// TwinCAT 3 PLC project Library
// Title: MTP
// Company: Zerlauth
// Author: Peter Zerlauth
// ProjectVersion: 0.0.0.0
// Description: Module Type Package MTP
// ProgramVersion: 3.1.4024.0
// libraries:
//   Tc2_Standard, * (Beckhoff Automation GmbH)
//   Tc2_System, * (Beckhoff Automation GmbH)
//   Tc2_Utilities, * (Beckhoff Automation GmbH)
// project tree:
//   Component/Event/ E_Event.TcDUT, FB_Event.TcPOU, I_Event.TcIO, ST_Event.TcDUT
//   Component/ E_Request.TcDUT, E_State.TcDUT, FB_Component.TcPOU, I_Component.TcIO, ST_Component.TcDUT (not stored)
//   Component/Info/ FB_Info.TcPOU, I_Info.TcIO (not stored)
//   Component/Observer/ FB_Observer.TcPOU, I_Observer.TcIO
//   List/ FB_ListComponent.TcPOU, FB_ListObject.TcPOU, FB_ListString.TcPOU, I_ListComponent.TcIO, I_ListObject.TcIO, I_ListString.TcIO (not stored)
//   Logger/ FB_ListLogger.TcPOU, I_Logger.TcIO
//   Object/ I_Object.TcIO
//   Sequence/ FB_Sequence.TcPOU (not stored), I_Sequence.TcIO (not stored)
// (motion and I/O tree: see PLC project example)
// real-time tasks:
//   TASK plcTask1: cycle T#1000ms, priority 20, ADS port 350

// ---- Component/Event/E_Event.TcDUT
{attribute 'qualified_only'}
{attribute 'strict'}
TYPE E_Event :
(
	Verbose			:= 0,
	Debug			:= 1,
	Information		:= 2,
	Warning			:= 3,
	Error			:= 4
);
END_TYPE

// ---- Component/Event/ST_Event.TcDUT
TYPE ST_Event :
STRUCT
	Timestamp:   	ULINT;
	ID:				UDINT;
	Message:		STRING(255);
	Arguments:		STRING(255);
END_STRUCT
END_TYPE

// ---- Component/E_Request.TcDUT
{attribute 'qualified_only'}
{attribute 'strict'}
TYPE E_Request :
(
    Undefined   := 0,
	Reset       := 1,
    Start       := 2,
    Pause       := 4,	
    Hold      	:= 8,
	Complete	:= 16,	
    Stop        := 32,
	Abort       := 64
);
END_TYPE

// ---- Component/E_State.TcDUT
{attribute 'qualified_only'}
{attribute 'strict'}
TYPE E_State :
(
	Undefined		:= 0,
	Clearing		:= 1,
	Stopped			:= 2,
	Starting		:= 3,
	Idle			:= 4,
	Suspend			:= 5,
	Execute			:= 6,
	Stopping		:= 7,
	Aborting		:= 8,
	Aborted			:= 9,
	Holding			:= 10,
	Held			:= 11,
	Unholding		:= 12,
	Suspending		:= 13,
	Unsuspending	:= 14,
	Resetting		:= 15,
	Completing		:= 16,
	Complete		:= 17
);
END_TYPE

// ---- Component/Event/I_Event.TcIO
INTERFACE I_Event EXTENDS I_Object

METHOD PUBLIC M_Abort : BOOL
VAR_INPUT
	Message:				STRING(255);
	ID:						UDINT;
END_VAR
END_METHOD

METHOD PUBLIC M_Debug : BOOL
VAR_INPUT
	Message:				STRING(255);
END_VAR
END_METHOD

METHOD PUBLIC M_Information : BOOL
VAR_INPUT
	Message:				STRING(255);
	ID:						UDINT;
END_VAR
END_METHOD

METHOD PUBLIC M_Stop : BOOL
VAR_INPUT
	Message:				STRING(255);
	ID:						UDINT;
END_VAR
END_METHOD

METHOD PUBLIC M_Warning : BOOL
VAR_INPUT
	Message:				STRING(255);
	ID:						UDINT;
END_VAR
END_METHOD

PROPERTY PUBLIC P_Logger : I_Logger
GET
END_GET
SET
END_SET
END_PROPERTY

END_INTERFACE

// ---- Component/I_Component.TcIO
INTERFACE I_Component EXTENDS I_Object

METHOD PUBLIC M_Request : BOOL
VAR_INPUT
	eRequest:	E_Request;
END_VAR
END_METHOD

PROPERTY PUBLIC P_Event : I_Event
GET
END_GET
END_PROPERTY

PROPERTY PUBLIC P_Info : I_Info
GET
END_GET
END_PROPERTY

PROPERTY PUBLIC P_Observer : I_Observer
GET
END_GET
END_PROPERTY

END_INTERFACE

// ---- Component/Observer/I_Observer.TcIO
INTERFACE I_Observer

METHOD M_Attach : BOOL
VAR_INPUT
	Object: 	I_Component;
END_VAR
END_METHOD

METHOD M_Detach : BOOL
VAR_INPUT
	Object: 	I_Component;
END_VAR
END_METHOD

METHOD M_Notify : BOOL
VAR_INPUT
	eRequest:		E_Request;
END_VAR
END_METHOD

END_INTERFACE

// ---- List/I_ListComponent.TcIO
INTERFACE I_ListComponent

METHOD M_Add : BOOL
VAR_INPUT
	Object: 	I_Component;
END_VAR
END_METHOD

METHOD M_Clear : BOOL
END_METHOD

METHOD M_Find : DINT
VAR_INPUT
	Object: 	I_Component;
END_VAR
END_METHOD

METHOD M_Index : I_Component
VAR_INPUT
	Index: 	DINT;
END_VAR
END_METHOD

METHOD M_Remove : BOOL
VAR_INPUT
	Object: 	I_Component;
END_VAR
END_METHOD

METHOD PUBLIC M_Request : BOOL
VAR_INPUT
	eRequest:		E_Request;
END_VAR
END_METHOD

PROPERTY P_Length : DINT
GET
END_GET
END_PROPERTY

END_INTERFACE

// ---- List/I_ListObject.TcIO
INTERFACE I_ListObject

METHOD M_Add : BOOL
VAR_INPUT
	Object: 	I_Object;
END_VAR
END_METHOD

METHOD M_Clear : BOOL
END_METHOD

METHOD M_Find : DINT
VAR_INPUT
	Object: 	I_Object;
END_VAR
END_METHOD

METHOD M_Index : I_Object
VAR_INPUT
	Index: 	DINT;
END_VAR
END_METHOD

METHOD M_Remove : BOOL
VAR_INPUT
	Object: 	I_Object;
END_VAR
END_METHOD

PROPERTY P_Length : DINT
GET
END_GET
END_PROPERTY

END_INTERFACE

// ---- Logger/I_Logger.TcIO
INTERFACE I_Logger EXTENDS I_Object

METHOD PUBLIC M_Log
VAR_INPUT
	stEvent:		ST_Event;
END_VAR
END_METHOD

END_INTERFACE

// ---- Object/I_Object.TcIO
INTERFACE I_Object EXTENDS __SYSTEM.IQueryInterface

END_INTERFACE

// ---- Component/Event/FB_Event.TcPOU
FUNCTION_BLOCK FB_Event EXTENDS FB_ListString IMPLEMENTS I_Event
VAR_INPUT
END_VAR
VAR_OUTPUT
END_VAR
VAR
	iParent:			I_Component;
	iLogger:			I_Logger;
	stEvent:			ST_Event;
END_VAR

SUPER^();

METHOD FB_init : BOOL
VAR_INPUT
	bInitRetains : BOOL; // if TRUE, the retain variables are initialized (warm start / cold start)
	bInCopyCode : BOOL;  // if TRUE, the instance afterwards gets moved into the copy code (online change)
	iParent:			I_Component;
END_VAR
THIS^.iParent:= iParent;
END_METHOD

METHOD PUBLIC M_Abort : BOOL
VAR_INPUT
	Message:				STRING(255);
	ID:						UDINT;
END_VAR
stEvent.Source:= iParent;
stEvent.EventType:= E_Event.Error;
stEvent.Timestamp:= F_GetSystemTime();
stEvent.ID:= ID;
stEvent.Message:= Message;
stEvent.Arguments:= M_Arguments();
stEvent.Active:= TRUE;

iParent.M_Request(E_Request.Abort);
IF iLogger <> 0 THEN
	iLogger.M_Log(stEvent);
END_IF

M_Clear();
END_METHOD

METHOD INTERNAL M_Arguments : STRING(255)
VAR_INPUT
END_VAR
VAR
	nIndex:			INT;
END_VAR
WHILE nIndex < nLength DO
	M_Arguments:= Concat(Concat(M_Arguments, pList[nIndex]), '$N');
	nIndex:= nIndex + 1;
END_WHILE
END_METHOD

METHOD PUBLIC M_Debug : BOOL
VAR_INPUT
	Message:				STRING(255);
END_VAR
END_METHOD

METHOD PUBLIC M_Information : BOOL
VAR_INPUT
	Message:				STRING(255);
	ID:						UDINT;
END_VAR
END_METHOD

METHOD PUBLIC M_Stop : BOOL
VAR_INPUT
	Message:				STRING(255);
	ID:						UDINT;
END_VAR

stEvent.Timestamp:= F_GetSystemTime();
stEvent.Message:= Message;
stEvent.ID:= ID;
stEvent.Arguments:= M_Arguments();
iParent.M_Request(E_Request.Stop);
M_Clear();
END_METHOD

METHOD PUBLIC M_Warning : BOOL
VAR_INPUT
	Message:				STRING(255);
	ID:						UDINT;
END_VAR
END_METHOD

PROPERTY PUBLIC P_Logger : I_Logger
GET
P_Logger:= iLogger;
END_GET
SET
iLogger:= P_Logger;
END_SET
END_PROPERTY

END_FUNCTION_BLOCK

// ---- List/FB_ListString.TcPOU
{attribute 'no_explicit_call'} 
FUNCTION_BLOCK FB_ListString IMPLEMENTS I_ListString
VAR
	pList: 			POINTER TO STRING(255);
	nLength:		DINT;
	aList:			POINTER TO POINTER TO ARRAY [0..100] OF STRING(255):=ADR(pList);
END_VAR

METHOD FB_exit : BOOL
VAR_INPUT
	bInCopyCode : BOOL; // if TRUE, the exit method is called for exiting an instance that is copied afterwards (online change).
END_VAR
M_Clear();
END_METHOD

METHOD PUBLIC M_Add : BOOL
VAR_INPUT
	Object: 	STRING(255);
END_VAR
VAR
	pOldList: 	POINTER TO STRING(255);
END_VAR
IF Object <> '' THEN
	// First Item
	IF pList = 0 THEN
		nLength:= nLength + 1;
		pList:= __NEW(STRING(255),DINT_TO_UDINT(nLength));
	ELSE
		// Item already in List
		IF M_Find(Object) = -1 THEN
			// backup 
			pOldList:= pList;
			// new Length
			nLength:= nLength + 1;
			// new pointer
			pList:= __NEW(STRING(255),DINT_TO_UDINT(nLength));
			// restore
			Memcpy(pList,pOldList, SIZEOF(STRING(255))*DINT_TO_UDINT(nLength -1));
			// delete old
			__DELETE(pOldList);
		ELSE
			M_Add:= FALSE;	
			RETURN;
		END_IF
	END_IF
	IF pList = 0 THEN
		RETURN;
	END_IF
	// add new Object
	pList[nLength-1]:= Object;
	M_Add:= TRUE;
ELSE
	M_Add:= FALSE;	
END_IF
END_METHOD

METHOD PUBLIC M_Clear : BOOL
IF pList <> 0 THEN
	nLength:= 0;
	__DELETE(pList);
END_IF
M_Clear:= True;
END_METHOD

METHOD PUBLIC M_Find : DINT
VAR_INPUT
	Object: 	STRING(255);
END_VAR
VAR
	nIndex: 	UINT;
END_VAR
// Object already in List
M_Find := -1;
WHILE nIndex < nLength DO
    IF (pList[nIndex] = Object) THEN
        M_Find := nIndex;
        RETURN;
    END_IF
	nIndex := nIndex + 1;
END_WHILE
END_METHOD

METHOD PUBLIC M_Index : STRING(255)
VAR_INPUT
	Index: 	DINT;
END_VAR
IF Index <= nLength THEN
	M_Index:= pList[Index];
END_IF
END_METHOD

METHOD PUBLIC M_Remove : BOOL
VAR_INPUT
	Object: 	STRING(255);
END_VAR
VAR
	pOldList:			POINTER TO STRING(255);
	nPosition: 			DINT;
END_VAR
IF Object <> '' THEN
	// First Item
	IF nLength >= 0 THEN
		// Item already in List
		nPosition:= M_Find(Object);
		IF nPosition <> -1 THEN
			// backup 
			pOldList:= pList;
			// new Length
			nLength:= nLength -1;
			// new pointer
			pList:= __NEW(POINTER TO I_Object,DINT_TO_UDINT(nLength));
			// restore lower part
			Memcpy(pList,pOldList, SIZEOF(STRING(255)) * DINT_TO_UDINT(nPosition));
			//pList[nPosition]:= iObject;
			Memcpy(pList + (SIZEOF(STRING(255))*nPosition),pOldList + (SIZEOF(STRING(255))*(nPosition + 1)), SIZEOF(STRING(255)) * DINT_TO_UDINT(nLength - nPosition));
			// delete old
			__DELETE(pOldList);
		ELSE
			M_Remove:= FALSE;	
			RETURN;
		END_IF
	ELSE
		M_Remove:= FALSE;	
		RETURN;
	END_IF
	M_Remove:= TRUE;
ELSE
	M_Remove:= FALSE;	
END_IF
END_METHOD

PROPERTY PUBLIC P_Length : DINT
GET
P_Length:= nLength;
END_GET
END_PROPERTY

END_FUNCTION_BLOCK

// ---- Component/FB_Component.TcPOU
{attribute 'reflection'} 
FUNCTION_BLOCK FB_Component IMPLEMENTS I_Component
VAR_INPUT
	fbInfo:						FB_Info(sInstancePath, eState);
	fbObserver:					FB_Observer;
	fbEvent:					FB_Event(THIS^);
END_VAR
VAR_OUTPUT
END_VAR
VAR
	stComponent:				ST_Component;
    {attribute 'hide'}
	{attribute 'instance-path'} 
    {attribute 'noinit'}
    sInstancePath:				STRING(255);	
	eRequest:					E_Request;
	eState:						E_State;
    {attribute 'hide'}
	eStatePrevious:				E_State;
END_VAR

fbInfo();
fbObserver();
fbEvent();

// Handle Module Type Package states
CASE eState OF
	E_State.Undefined:
		IF M_Initialise() THEN
			eState:= E_State.Idle;					
		END_IF
		
	E_State.Resetting:
		CASE eRequest OF
			E_Request.Stop:
				fbObserver.M_Notify(E_Request.Stop);
				eState:= E_State.Stopping;					
			E_Request.Abort:
				fbObserver.M_Notify(E_Request.Abort);
				eState:= E_State.Aborting;						
		END_CASE	
		IF M_Resetting() THEN
			eState:= E_State.Idle;
		END_IF
		
	E_State.Idle:
		CASE eRequest OF
			E_Request.Start:
				eState:= E_State.Starting;
			E_Request.Stop:
				fbObserver.M_Notify(E_Request.Stop);
				eState:= E_State.Stopping;					
			E_Request.Abort:
				fbObserver.M_Notify(E_Request.Abort);
				eState:= E_State.Aborting;						
		END_CASE
		M_Idle();
		
	E_State.Starting:
		CASE eRequest OF
			E_Request.Stop:
				fbObserver.M_Notify(E_Request.Stop);
				eState:= E_State.Stopping;					
			E_Request.Abort:
				fbObserver.M_Notify(E_Request.Abort);
				eState:= E_State.Aborting;						
		END_CASE	
		IF M_Starting() THEN
			eState:= E_State.Execute;	
		END_IF		

	E_State.Execute:
		CASE eRequest OF
			E_Request.Pause:
				eState:= E_State.Pausing;		
			E_Request.Hold:
				eState:= E_State.Holding;		
			E_Request.Stop:
				fbObserver.M_Notify(E_Request.Stop);
				eState:= E_State.Stopping;					
			E_Request.Abort:
				fbObserver.M_Notify(E_Request.Abort);
				eState:= E_State.Aborting;						
		END_CASE	
		IF M_Execute() THEN
			CASE eRequest OF
				E_Request.Complete:
					eState:= E_State.Completing;					
			END_CASE	
		END_IF
		
	E_State.Stopping:
		CASE eRequest OF	
			E_Request.Abort:
				eState:= E_State.Aborting;						
		END_CASE	
		IF M_Stopping() THEN
			eState:= E_State.Stopped;	
		END_IF

	E_State.Stopped:
		IF M_Stopped() THEN
			CASE eRequest OF
				E_Request.Reset:
					eState:= E_State.Resetting;					
			END_CASE		
		END_IF
		
	E_State.Aborting:
		IF M_Aborting() THEN
			eState:= E_State.Aborted;	
		END_IF
		
	E_State.Aborted:
		IF M_Aborted() THEN
			CASE eRequest OF
				E_Request.Reset:
					eState:= E_State.Resetting;					
			END_CASE	
		END_IF
		
	E_State.Pausing:
		CASE eRequest OF
			E_Request.Stop:
				fbObserver.M_Notify(E_Request.Stop);
				eState:= E_State.Stopping;					
			E_Request.Abort:
				fbObserver.M_Notify(E_Request.Abort);
				eState:= E_State.Aborting;						
		END_CASE	
		IF M_Pausing() THEN
			eState:= E_State.Paused;
		END_IF
	
	E_State.Paused:
		CASE eRequest OF
			E_Request.Stop:
				fbObserver.M_Notify(E_Request.Stop);
				eState:= E_State.Stopping;					
			E_Request.Abort:
				fbObserver.M_Notify(E_Request.Abort);
				eState:= E_State.Aborting;						
		END_CASE	
		IF M_Paused() THEN
			eState:= E_State.Resuming;			
		END_IF	
		
	E_State.Resuming:
		CASE eRequest OF
			E_Request.Stop:
				fbObserver.M_Notify(E_Request.Stop);
				eState:= E_State.Stopping;					
			E_Request.Abort:
				fbObserver.M_Notify(E_Request.Abort);
				eState:= E_State.Aborting;					
		END_CASE
		IF M_Resuming() THEN
			eState:= E_State.Execute;
		END_IF

	E_State.Holding:
		CASE eRequest OF
			E_Request.Stop:
				fbObserver.M_Notify(E_Request.Stop);
				eState:= E_State.Stopping;					
			E_Request.Abort:
				fbObserver.M_Notify(E_Request.Abort);
				eState:= E_State.Aborting;						
		END_CASE
		IF M_Holding() THEN
			eState:= E_State.Held;
		END_IF

	E_State.Held:
		CASE eRequest OF
			E_Request.Stop:
				fbObserver.M_Notify(E_Request.Stop);
				eState:= E_State.Stopping;					
			E_Request.Abort:
				fbObserver.M_Notify(E_Request.Abort);
				eState:= E_State.Aborting;					
		END_CASE
		IF M_Held() THEN
			eState:= E_State.Unholding;			
		END_IF	
		
	E_State.Unholding:
		CASE eRequest OF
			E_Request.Stop:
				fbObserver.M_Notify(E_Request.Stop);
				eState:= E_State.Stopping;					
			E_Request.Abort:
				fbObserver.M_Notify(E_Request.Abort);
				eState:= E_State.Aborting;							
		END_CASE
		IF M_Unholding() THEN
			eState:= E_State.Execute;
		END_IF
		
	E_State.Completing:
		CASE eRequest OF
			E_Request.Stop:
				fbObserver.M_Notify(E_Request.Stop);
				eState:= E_State.Stopping;					
			E_Request.Abort:
				fbObserver.M_Notify(E_Request.Abort);
				eState:= E_State.Aborting;						
		END_CASE
		IF M_Completing() THEN
			eState:= E_State.Completed;
		END_IF
		
	E_State.Completed:
		CASE eRequest OF
			E_Request.Stop:
				fbObserver.M_Notify(E_Request.Stop);
				eState:= E_State.Stopping;					
			E_Request.Abort:
				fbObserver.M_Notify(E_Request.Abort);
				eState:= E_State.Aborting;						
		END_CASE
		IF M_Completed() THEN
			CASE eRequest OF
				E_Request.Reset:	
					eState:= E_State.Resetting;
			END_CASE
		END_IF
	
END_CASE

// Detect state changed
IF eStatePrevious <> eState THEN
	eStatePrevious:= eState;
	M_StateChanged();
END_IF
eRequest:= E_Request.Undefined;

METHOD PROTECTED M_Aborted : BOOL
VAR_INPUT
END_VAR
// State Aborted
M_Aborted:= True;
END_METHOD

METHOD PROTECTED M_Aborting : BOOL
VAR_INPUT
END_VAR
// State Aborting
M_Aborting:= True;
END_METHOD

METHOD PROTECTED M_Completed : BOOL
VAR_INPUT
END_VAR
// State Complete
M_Completed:= TRUE;
END_METHOD

METHOD PROTECTED M_Completing : BOOL
VAR_INPUT
END_VAR
// State Completing
M_Completing:= True;
END_METHOD

METHOD PROTECTED M_Execute : BOOL
VAR_INPUT
END_VAR
// State Execute
M_Execute:= TRUE;
END_METHOD

METHOD PROTECTED M_Held : BOOL
VAR_INPUT
END_VAR
// State Held
M_Held:= TRUE;
END_METHOD

METHOD PROTECTED M_Holding : BOOL
VAR_INPUT
END_VAR
// State Holding
M_Holding:= True;
END_METHOD

METHOD PROTECTED M_Idle : BOOL
VAR_INPUT
END_VAR
// State Idle
END_METHOD

METHOD PROTECTED M_Initialise : BOOL;
VAR_INPUT
END_VAR
// State Undefined
M_Initialise:= True;
END_METHOD

METHOD PROTECTED M_Paused : BOOL
VAR_INPUT
END_VAR
// State Held
M_Paused:= TRUE;
END_METHOD

METHOD PROTECTED M_Pausing : BOOL
VAR_INPUT
END_VAR
// State Holding
M_Pausing:= True;
END_METHOD

METHOD PUBLIC M_Request : BOOL
VAR_INPUT
	eRequest:	E_Request;
END_VAR
THIS^.eRequest:= eRequest;
CASE eRequest OF
	E_Request.Undefined:
		M_Request:= TRUE;
    E_Request.Start:
		M_Request:= eState = E_State.Execute;
    E_Request.Pause:
		M_Request:= eState = E_State.Paused;
    E_Request.Hold:
		M_Request:= eState = E_State.Held;
	E_Request.Complete:
		M_Request:= eState = E_State.Completed;	
    E_Request.Stop:
		M_Request:= eState = E_State.Stopped;	
	E_Request.Abort:
		M_Request:= eState = E_State.Aborted;	
	E_Request.Reset:
		M_Request:= eState = E_State.Idle;		

END_CASE
END_METHOD

METHOD PROTECTED M_Resetting : BOOL
VAR_INPUT
END_VAR
// State Resetting
M_Resetting:= True;
END_METHOD

METHOD PROTECTED M_Resuming : BOOL
VAR_INPUT
END_VAR
// State Holding
M_Resuming:= True;
END_METHOD

METHOD PROTECTED M_Starting : BOOL
VAR_INPUT
END_VAR
// State Starting
M_Starting:= True;
END_METHOD

METHOD PROTECTED M_StateChanged : BOOL
VAR_INPUT
END_VAR
END_METHOD

METHOD PROTECTED M_Stopped : BOOL
VAR_INPUT
END_VAR
// State Stopped
M_Stopped:= True;
END_METHOD

METHOD PROTECTED M_Stopping : BOOL
VAR_INPUT
END_VAR
// State Stopping
M_Stopping:= True;
END_METHOD

METHOD PROTECTED M_Unholding : BOOL
VAR_INPUT
END_VAR
// State Holding
M_Unholding:= True;
END_METHOD

PROPERTY PUBLIC P_Event : I_Event
GET
P_Event:= fbEvent;
END_GET
END_PROPERTY

PROPERTY PUBLIC P_Info : I_Info
GET
P_Info:= fbInfo;
END_GET
END_PROPERTY

PROPERTY PUBLIC P_Observer : I_Observer
GET
P_Observer:= fbObserver;
END_GET
END_PROPERTY

END_FUNCTION_BLOCK

// ---- Component/Info/FB_Info.TcPOU
FUNCTION_BLOCK PUBLIC FB_Info IMPLEMENTS I_Info
VAR_INPUT
END_VAR
VAR_OUTPUT
END_VAR
VAR
    sInstancePath:				REFERENCE TO STRING(255);
	eState:						REFERENCE TO E_State;
	fbReadSymInfo: 				PLC_ReadSymInfoByNameEx;
	nIndex:						DINT;
END_VAR
VAR_STAT
	nCycle: 					UDINT;
	nTimestamp: 				ULINT;
END_VAR

GETCURTASKINDEXEX(GETCURTASKINDEXEX => nIndex);
IF nCycle <> TwinCAT_SystemInfoVarList._TaskInfo[nIndex].CycleCount THEN
	nCycle:= TwinCAT_SystemInfoVarList._TaskInfo[nIndex].CycleCount;
	nTimestamp:= F_GetSystemTime();
END_IF

fbReadSymInfo(
	NETID:= , 
	PORT:= , 
	SYMNAME:= , 
	START:= , 
	TMOUT:= , 
	BUSY=> , 
	ERR=> , 
	ERRID=> , 
	SYMINFO=> , 
	OVTYPE=> , 
	OVCOMMENT=> );

METHOD FB_init : BOOL
VAR_INPUT
	bInitRetains : BOOL; // if TRUE, the retain variables are initialized (warm start / cold start)
	bInCopyCode : BOOL;  // if TRUE, the instance afterwards gets moved into the copy code (online change)
	sInstancePath:			REFERENCE TO STRING(255);
	eState:					REFERENCE TO E_State;
	
END_VAR
THIS^.sInstancePath REF= sInstancePath;
THIS^.eState REF= eState;
M_Initialize();
END_METHOD

METHOD PROTECTED M_Initialize
VAR_INPUT
END_VAR
VAR
    sName:				STRING(255);
    nPosition:			INT;
END_VAR
sName := CONCAT(TwinCAT_SystemInfoVarList._AppInfo.ProjectName, '.');

nPosition := FIND(sInstancePath, sName);
IF nPosition > 0 THEN
    fbReadSymInfo.SYMNAME:= DELETE(sInstancePath, nPosition-1 + LEN(sName), 1);
END_IF

nPosition := FIND(fbReadSymInfo.SYMNAME, sName);

IF nPosition > 0 THEN
    fbReadSymInfo.SYMNAME:= DELETE(fbReadSymInfo.SYMNAME, nPosition - 1 + LEN(sName), 1);
END_IF

fbReadSymInfo.PORT:= TwinCAT_SystemInfoVarList._AppInfo.AdsPort;
fbReadSymInfo.START:= TRUE;
END_METHOD

PROPERTY PUBLIC P_Class : String(255)
GET
P_Class:= fbReadSymInfo.SYMINFO.symDataType;
END_GET
END_PROPERTY

PROPERTY PUBLIC P_Comment : String(255)
GET
P_Comment:= fbReadSymInfo.SYMINFO.symComment;
END_GET
END_PROPERTY

PROPERTY PUBLIC P_Instance : String(255)
GET
P_Instance:= fbReadSymInfo.SYMNAME;
END_GET
END_PROPERTY

PROPERTY PUBLIC P_State : E_State
GET
P_State:= eState;
END_GET
END_PROPERTY

PROPERTY PUBLIC P_Timestamp : ULINT
GET
P_Timestamp:= nTimestamp;
END_GET
END_PROPERTY

END_FUNCTION_BLOCK

// ---- Component/Observer/FB_Observer.TcPOU
{attribute 'no_explicit_call'} 
FUNCTION_BLOCK PUBLIC FB_Observer IMPLEMENTS I_Observer
VAR
	pList: 			POINTER TO I_Component;
	nLength:		DINT;
	aList:			POINTER TO POINTER TO ARRAY [0..100] OF I_Component:=ADR(pList);
END_VAR

METHOD FB_exit : BOOL
VAR_INPUT
	bInCopyCode : BOOL; // if TRUE, the exit method is called for exiting an instance that is copied afterwards (online change).
END_VAR
M_Clear();
END_METHOD

METHOD M_Attach : BOOL
VAR_INPUT
	Object: 	I_Component;
END_VAR
VAR
	pOldList: 	POINTER TO I_Component;
END_VAR
IF Object <> 0 THEN
	// First Item
	IF pList = 0 THEN
		nLength:= nLength + 1;
		pList:= __NEW(POINTER TO I_Component,DINT_TO_UDINT(nLength));
	ELSE
		// Item already in List
		IF M_Find(Object) = -1 THEN
			// backup 
			pOldList:= pList;
			// new Length
			nLength:= nLength + 1;
			// new pointer
			pList:= __NEW(POINTER TO I_Component,DINT_TO_UDINT(nLength));
			// restore
			Memcpy(pList,pOldList, SIZEOF(POINTER TO I_Component)*DINT_TO_UDINT(nLength -1));
			// delete old
			__DELETE(pOldList);
		ELSE
			M_Attach:= FALSE;	
			RETURN;
		END_IF
	END_IF
	IF pList = 0 THEN
		RETURN;
	END_IF
	// add new Object
	pList[nLength-1]:= Object;
	M_Attach:= TRUE;
ELSE
	M_Attach:= FALSE;	
END_IF
END_METHOD

METHOD M_Clear
IF pList <> 0 THEN
	nLength:= 0;
	__DELETE(pList);
END_IF
END_METHOD

METHOD M_Detach : BOOL
VAR_INPUT
	Object: 	I_Component;
END_VAR
VAR
	pOldList:			POINTER TO I_Component;
	nPosition: 			DINT;
END_VAR
IF Object <> 0 THEN
	// First Item
	IF nLength >= 0 THEN
		// Item already in List
		nPosition:= M_Find(Object);
		IF nPosition <> -1 THEN
			// backup 
			pOldList:= pList;
			// new Length
			nLength:= nLength -1;
			// new pointer
			pList:= __NEW(POINTER TO I_Component,DINT_TO_UDINT(nLength));
			// restore lower part
			Memcpy(pList,pOldList, SIZEOF(POINTER TO I_Component) * DINT_TO_UDINT(nPosition));
			//pList[nPosition]:= iObject;
			Memcpy(pList + (SIZEOF(POINTER TO I_Component)*nPosition),pOldList + (SIZEOF(POINTER TO I_Component)*(nPosition + 1)), SIZEOF(POINTER TO I_Component) * DINT_TO_UDINT(nLength - nPosition));
			// delete old
			__DELETE(pOldList);
		ELSE
			M_Detach:= FALSE;	
			RETURN;
		END_IF
	ELSE
		M_Detach:= FALSE;	
		RETURN;
	END_IF
	M_Detach:= TRUE;
ELSE
	M_Detach:= FALSE;	
END_IF
END_METHOD

METHOD M_Find : DINT
VAR_INPUT
	Object: 	I_Component;
END_VAR
VAR
	nIndex: 	UINT;
END_VAR
// Object already in List
M_Find := -1;
WHILE nIndex < nLength DO
    IF (pList[nIndex] = Object) THEN
        M_Find := nIndex;
        RETURN;
    END_IF
	nIndex := nIndex + 1;
END_WHILE
END_METHOD

METHOD M_Index : I_Component
VAR_INPUT
	Index: 	DINT;
END_VAR
IF Index <= nLength THEN
	M_Index:= pList[Index];
END_IF
END_METHOD

METHOD M_Notify : BOOL
VAR_INPUT
	eRequest:		E_Request;
END_VAR

VAR
	nIndex: 	INT;
END_VAR
WHILE nIndex < nLength DO
	pList[nIndex].M_Request(eRequest);
	nIndex:= nIndex + 1; 
END_WHILE
END_METHOD

PROPERTY P_Length : DINT
GET
P_Length:= nLength;
END_GET
END_PROPERTY

END_FUNCTION_BLOCK

// ---- List/FB_ListComponent.TcPOU
{attribute 'no_explicit_call'} 
FUNCTION_BLOCK FB_ListComponent IMPLEMENTS I_ListComponent
VAR
	nLength:		DINT;
	aList:			POINTER TO POINTER TO ARRAY [0..100] OF I_Component:=ADR(pList);
	pList: 			POINTER TO I_Component;
END_VAR

METHOD FB_exit : BOOL
VAR_INPUT
	bInCopyCode : BOOL; // if TRUE, the exit method is called for exiting an instance that is copied afterwards (online change).
END_VAR
M_Clear();
END_METHOD

METHOD M_Add : BOOL
VAR_INPUT
	Object: 	I_Component;
END_VAR
VAR
	pOldList: 	POINTER TO I_Component;
END_VAR
IF Object <> 0 THEN
	// First Item
	IF pList = 0 THEN
		nLength:= nLength + 1;
		pList:= __NEW(POINTER TO I_Component,DINT_TO_UDINT(nLength));
	ELSE
		// Item already in List
		IF M_Find(Object) = -1 THEN
			// backup 
			pOldList:= pList;
			// new Length
			nLength:= nLength + 1;
			// new pointer
			pList:= __NEW(POINTER TO I_Component,DINT_TO_UDINT(nLength));
			// restore
			Memcpy(pList,pOldList, SIZEOF(POINTER TO I_Component)*DINT_TO_UDINT(nLength -1));
			// delete old
			__DELETE(pOldList);
		ELSE
			M_Add:= FALSE;	
			RETURN;
		END_IF
	END_IF
	IF pList = 0 THEN
		RETURN;
	END_IF
	// add new Object
	pList[nLength-1]:= Object;
	M_Add:= TRUE;
ELSE
	M_Add:= FALSE;	
END_IF
END_METHOD

METHOD PUBLIC M_Add2 : BOOL
VAR_INPUT
	Parent: 	I_Component;
	Object: 	I_Component;
END_VAR
M_Add(Object);
Parent.P_Event.P_Observer.M_Attach(Object);
END_METHOD

METHOD M_Clear : BOOL
// Clear
IF pList <> 0 THEN
	nLength:= 0;
	__DELETE(pList);
END_IF
M_Clear:= TRUE;
END_METHOD

METHOD M_Find : DINT
VAR_INPUT
	Object: 	I_Component;
END_VAR
VAR
	nIndex: 	UINT;
END_VAR
// Find
M_Find := -1;
WHILE nIndex < nLength DO
    IF (pList[nIndex] = Object) THEN
        M_Find := nIndex;
        RETURN;
    END_IF
	nIndex := nIndex + 1;
END_WHILE
END_METHOD

METHOD M_Index : I_Component
VAR_INPUT
	Index: 	DINT;
END_VAR
// Index
IF Index <= nLength THEN
	M_Index:= pList[Index];
END_IF
END_METHOD

METHOD M_Remove : BOOL
VAR_INPUT
	Object: 	I_Component;
END_VAR
VAR
	pOldList:			POINTER TO I_Component;
	nPosition: 			DINT;
END_VAR
// Remove
IF Object <> 0 THEN
	// First Item
	IF nLength >= 0 THEN
		// Item already in List
		nPosition:= M_Find(Object);
		IF nPosition <> -1 THEN
			// backup 
			pOldList:= pList;
			// new Length
			nLength:= nLength -1;
			// new pointer
			pList:= __NEW(POINTER TO I_Component,DINT_TO_UDINT(nLength));
			// restore lower part
			Memcpy(pList,pOldList, SIZEOF(POINTER TO I_Object) * DINT_TO_UDINT(nPosition));
			//pList[nPosition]:= iObject;
			Memcpy(pList + (SIZEOF(POINTER TO I_Component)*nPosition),pOldList + (SIZEOF(POINTER TO I_Component)*(nPosition + 1)), SIZEOF(POINTER TO I_Component) * DINT_TO_UDINT(nLength - nPosition));
			// delete old
			__DELETE(pOldList);
		ELSE
			M_Remove:= FALSE;	
			RETURN;
		END_IF
	ELSE
		M_Remove:= FALSE;	
		RETURN;
	END_IF
	M_Remove:= TRUE;
ELSE
	M_Remove:= FALSE;	
END_IF
END_METHOD

METHOD PUBLIC M_Request : BOOL
VAR_INPUT
	eRequest:		E_Request;
END_VAR
VAR
	nIndex:			INT:= 0;
END_VAR
// Request
M_Request:= TRUE;
WHILE nIndex < P_Length DO
	M_Request:= M_Request AND M_Index(nIndex).M_Request(eRequest);
	nIndex:= nIndex + 1;
END_WHILE
END_METHOD

PROPERTY P_Length : DINT
GET
P_Length:= nLength;
END_GET
END_PROPERTY

END_FUNCTION_BLOCK

// ---- List/FB_ListObject.TcPOU
{attribute 'no_explicit_call'} 
FUNCTION_BLOCK FB_ListObject IMPLEMENTS I_ListObject
VAR
	pList: 			POINTER TO I_Object;
	nLength:		DINT;
	aList:			POINTER TO POINTER TO ARRAY [0..100] OF I_Object:=ADR(pList);
END_VAR

METHOD FB_exit : BOOL
VAR_INPUT
	bInCopyCode : BOOL; // if TRUE, the exit method is called for exiting an instance that is copied afterwards (online change).
END_VAR
M_Clear();
END_METHOD

METHOD M_Add : BOOL
VAR_INPUT
	Object: 	I_Object;
END_VAR
VAR
	pOldList: 	POINTER TO I_Object;
END_VAR
IF Object <> 0 THEN
	// First Item
	IF pList = 0 THEN
		nLength:= nLength + 1;
		pList:= __NEW(POINTER TO I_Object,DINT_TO_UDINT(nLength));
	ELSE
		// Item already in List
		IF M_Find(Object) = -1 THEN
			// backup 
			pOldList:= pList;
			// new Length
			nLength:= nLength + 1;
			// new pointer
			pList:= __NEW(POINTER TO I_Object,DINT_TO_UDINT(nLength));
			// restore
			Memcpy(pList,pOldList, SIZEOF(POINTER TO I_Object)*DINT_TO_UDINT(nLength -1));
			// delete old
			__DELETE(pOldList);
		ELSE
			M_Add:= FALSE;	
			RETURN;
		END_IF
	END_IF
	IF pList = 0 THEN
		RETURN;
	END_IF
	// add new Object
	pList[nLength-1]:= Object;
	M_Add:= TRUE;
ELSE
	M_Add:= FALSE;	
END_IF
END_METHOD

METHOD M_Clear : bool
IF pList <> 0 THEN
	nLength:= 0;
	__DELETE(pList);
END_IF
M_Clear:= True;
END_METHOD

METHOD M_Find : DINT
VAR_INPUT
	Object: 	I_Object;
END_VAR
VAR
	nIndex: 	UINT;
END_VAR
// Object already in List
M_Find := -1;
WHILE nIndex < nLength DO
    IF (pList[nIndex] = Object) THEN
        M_Find := nIndex;
        RETURN;
    END_IF
	nIndex := nIndex + 1;
END_WHILE
END_METHOD

METHOD M_Index : I_Object
VAR_INPUT
	Index: 	DINT;
END_VAR
IF Index <= nLength THEN
	M_Index:= pList[Index];
END_IF
END_METHOD

METHOD M_Remove : BOOL
VAR_INPUT
	Object: 	I_Object;
END_VAR
VAR
	pOldList:			POINTER TO I_Object;
	nPosition: 			DINT;
END_VAR
IF Object <> 0 THEN
	// First Item
	IF nLength >= 0 THEN
		// Item already in List
		nPosition:= M_Find(Object);
		IF nPosition <> -1 THEN
			// backup 
			pOldList:= pList;
			// new Length
			nLength:= nLength -1;
			// new pointer
			pList:= __NEW(POINTER TO I_Object,DINT_TO_UDINT(nLength));
			// restore lower part
			Memcpy(pList,pOldList, SIZEOF(POINTER TO I_Object) * DINT_TO_UDINT(nPosition));
			//pList[nPosition]:= iObject;
			Memcpy(pList + (SIZEOF(POINTER TO I_Object)*nPosition),pOldList + (SIZEOF(POINTER TO I_Object)*(nPosition + 1)), SIZEOF(POINTER TO I_Object) * DINT_TO_UDINT(nLength - nPosition));
			// delete old
			__DELETE(pOldList);
		ELSE
			M_Remove:= FALSE;	
			RETURN;
		END_IF
	ELSE
		M_Remove:= FALSE;	
		RETURN;
	END_IF
	M_Remove:= TRUE;
ELSE
	M_Remove:= FALSE;	
END_IF
END_METHOD

PROPERTY P_Length : DINT
GET
P_Length:= nLength;
END_GET
END_PROPERTY

END_FUNCTION_BLOCK

// ---- Logger/FB_ListLogger.TcPOU
{attribute 'no_explicit_call'} 
FUNCTION_BLOCK FB_ListLogger IMPLEMENTS I_Logger
VAR
	pList: 			POINTER TO I_Logger;
	nLength:		DINT;
	aList:			POINTER TO POINTER TO ARRAY [0..100] OF I_Logger:=ADR(pList);
END_VAR

METHOD FB_exit : BOOL
VAR_INPUT
	bInCopyCode : BOOL; // if TRUE, the exit method is called for exiting an instance that is copied afterwards (online change).
END_VAR
M_Clear();
END_METHOD

METHOD M_Add : BOOL
VAR_INPUT
	Object: 	I_Logger;
END_VAR
VAR
	pOldList: 	POINTER TO I_Logger;
END_VAR
IF Object <> 0 THEN
	// First Item
	IF pList = 0 THEN
		nLength:= nLength + 1;
		pList:= __NEW(POINTER TO I_Logger,DINT_TO_UDINT(nLength));
	ELSE
		// Item already in List
		IF M_Find(Object) = -1 THEN
			// backup 
			pOldList:= pList;
			// new Length
			nLength:= nLength + 1;
			// new pointer
			pList:= __NEW(POINTER TO I_Object,DINT_TO_UDINT(nLength));
			// restore
			Memcpy(pList,pOldList, SIZEOF(POINTER TO I_Logger)*DINT_TO_UDINT(nLength -1));
			// delete old
			__DELETE(pOldList);
		ELSE
			M_Add:= FALSE;	
			RETURN;
		END_IF
	END_IF
	IF pList = 0 THEN
		RETURN;
	END_IF
	// add new Object
	pList[nLength-1]:= Object;
	M_Add:= TRUE;
ELSE
	M_Add:= FALSE;	
END_IF
END_METHOD

METHOD M_Clear : bool
IF pList <> 0 THEN
	nLength:= 0;
	__DELETE(pList);
END_IF
M_Clear:= True;
END_METHOD

METHOD M_Find : DINT
VAR_INPUT
	Object: 	I_Logger;
END_VAR
VAR
	nIndex: 	UINT;
END_VAR
// Object already in List
M_Find := -1;
WHILE nIndex < nLength DO
    IF (pList[nIndex] = Object) THEN
        M_Find := nIndex;
        RETURN;
    END_IF
	nIndex := nIndex + 1;
END_WHILE
END_METHOD

METHOD M_Index : I_Logger
VAR_INPUT
	Index: 	DINT;
END_VAR
IF Index <= nLength THEN
	M_Index:= pList[Index];
END_IF
END_METHOD

METHOD PUBLIC M_Log
VAR_INPUT
	stEvent:		ST_Event;
END_VAR

VAR
	nIndex: INT;
END_VAR
WHILE nIndex < nLength DO
	M_Index(nIndex).M_Log(stEvent);
	nIndex:= nIndex +1;
END_WHILE
END_METHOD

METHOD M_Remove : BOOL
VAR_INPUT
	Object: 	I_Logger;
END_VAR
VAR
	pOldList:			POINTER TO I_Logger;
	nPosition: 			DINT;
END_VAR
IF Object <> 0 THEN
	// First Item
	IF nLength >= 0 THEN
		// Item already in List
		nPosition:= M_Find(Object);
		IF nPosition <> -1 THEN
			// backup 
			pOldList:= pList;
			// new Length
			nLength:= nLength -1;
			// new pointer
			pList:= __NEW(POINTER TO I_Logger,DINT_TO_UDINT(nLength));
			// restore lower part
			Memcpy(pList,pOldList, SIZEOF(POINTER TO I_Logger) * DINT_TO_UDINT(nPosition));
			//pList[nPosition]:= iObject;
			Memcpy(pList + (SIZEOF(POINTER TO I_Logger)*nPosition),pOldList + (SIZEOF(POINTER TO I_Logger)*(nPosition + 1)), SIZEOF(POINTER TO I_Logger) * DINT_TO_UDINT(nLength - nPosition));
			// delete old
			__DELETE(pOldList);
		ELSE
			M_Remove:= FALSE;	
			RETURN;
		END_IF
	ELSE
		M_Remove:= FALSE;	
		RETURN;
	END_IF
	M_Remove:= TRUE;
ELSE
	M_Remove:= FALSE;	
END_IF
END_METHOD

PROPERTY P_Length : DINT
GET
P_Length:= nLength;
END_GET
END_PROPERTY

END_FUNCTION_BLOCK
